(*
============================================================
PROGRAM: MAIN
============================================================

PURPOSE
  Top-level program that orchestrates all function blocks
  and manages the system data bus between GVLs.

EXECUTION ORDER (every PLC cycle)
  1. Initialise MQTT config from defaults (first scan only)
  2. Copy HMI inputs to GVL_System bus
  3. FB_SensorIO      — Read and scale analog sensor inputs
  4. FB_ValveControl  — Per-valve TC2_MC2 state machines (x3)
  5. Build timestamp string for MQTT and logging
  6. FB_MqttManager   — MQTT connection, publish, subscribe
  7. FB_CsvLogger     — Periodic CSV row logging
  8. Mirror runtime data to GVL_HMI for display
  9. Compute system health flags

DATA FLOW
  GVL_IO  --> FB_SensorIO --> GVL_System.Sensors
  GVL_HMI.HMI_* --> GVL_System.Valve[n] setpoints
  FB_MqttManager.rMqttValveSetpoint --> FB_ValveControl MQTT_Setpoint
  FB_ValveControl outputs --> GVL_System.Valve[n] status
  GVL_System.* --> GVL_HMI.ACT_* (for display)
  GVL_System.Valve + Sensors --> FB_MqttManager (outgoing JSON)
  GVL_System.Valve + Sensors --> FB_CsvLogger (CSV row)

LIBRARIES
  TC2_MC2, TF6701 / Tc3_IotBase, Tc2_System
============================================================
*)

PROGRAM MAIN
VAR
    // ── Function block instances ────────────────────────────────
    fbSensorIO      : FB_SensorIO;    //////Not Implemented currently
    fbValve1        : FB_ValveControl;
    fbValve2        : FB_ValveControl;
    fbValve3        : FB_ValveControl;
    fbCsvLogger     : FB_CsvLogger;
    fbMqttManager   : FB_MqttManager;

    // ── NC Axis references ──────────────────────────────────────
    // Each must be linked to an NC axis in TwinCAT I/O mapping.
    Axis_Valve1     : AXIS_REF;
    Axis_Valve2     : AXIS_REF;
    Axis_Valve3     : AXIS_REF;

    // ── Timestamp for MQTT JSON ──────────────────────────────────
    fbSysTime       : FB_LocalSystemTime;
    sTimestamp      : STRING(64);
    sTempStr        : STRING(8);

    // ── Whole-array buffers passed to FB_MqttManager ─────────────
    // TwinCAT does not allow per-element array assignment inside
    // an FB call's parameter list. Populate these arrays each
    // cycle, then pass them in a single assignment.
    aValveSetpoint  : ARRAY[1..3] OF REAL;
    aValveActual    : ARRAY[1..3] OF REAL;
    aValveSource    : ARRAY[1..3] OF STRING(8);

    // ── First-scan flag for MQTT default config load ─────────────
    bMqttConfigInit : BOOL := FALSE;
END_VAR

// ============================================================
// STEP 0 — ONE-TIME INITIALISATION
// On first scan, copy MQTT defaults from GVL_Config into the
// HMI-bound config struct. The operator can then edit any field
// from the HMI MQTT panel and click Apply to reconnect.
// ============================================================
IF NOT bMqttConfigInit THEN
    GVL_HMI.HMI_MQTT_Config.sBrokerAddress         := GVL_Config.MQTT_DEFAULT_BROKER_IP;
    GVL_HMI.HMI_MQTT_Config.nPort                  := GVL_Config.MQTT_DEFAULT_PORT;
    GVL_HMI.HMI_MQTT_Config.sClientId              := GVL_Config.MQTT_DEFAULT_CLIENT_ID;
    GVL_HMI.HMI_MQTT_Config.sUsername              := GVL_Config.MQTT_DEFAULT_USERNAME;
    GVL_HMI.HMI_MQTT_Config.sPassword              := GVL_Config.MQTT_DEFAULT_PASSWORD;
    GVL_HMI.HMI_MQTT_Config.sTopicPrefix           := GVL_Config.MQTT_DEFAULT_TOPIC_PREFIX;
    GVL_HMI.HMI_MQTT_Config.sMainTopic             := GVL_Config.MQTT_DEFAULT_MAIN_TOPIC;
    GVL_HMI.HMI_MQTT_Config.SubscribeTopic         := GVL_Config.MQTT_DEFAULT_SUB_TOPIC;
    GVL_HMI.HMI_MQTT_Config.tStatusPublishInterval := UDINT_TO_TIME(UINT_TO_UDINT(GVL_Config.MQTT_DEFAULT_PUBLISH_INTERVAL) * 1000);
    GVL_HMI.HMI_MQTT_Config.bUseStatusPublish      := TRUE;
   // bMqttConfigInit := TRUE;
END_IF


// ============================================================
// STEP 1 — COPY HMI SETPOINTS / RESETS INTO SYSTEM BUS
// ============================================================
GVL_System.Valve[1].HMI_Setpoint := GVL_HMI.HMI_Valve1_Setpoint;
GVL_System.Valve[1].Reset_Cmd    := GVL_HMI.HMI_Valve1_Reset;

GVL_System.Valve[2].HMI_Setpoint := GVL_HMI.HMI_Valve2_Setpoint;
GVL_System.Valve[2].Reset_Cmd    := GVL_HMI.HMI_Valve2_Reset;

GVL_System.Valve[3].HMI_Setpoint := GVL_HMI.HMI_Valve3_Setpoint;
GVL_System.Valve[3].Reset_Cmd    := GVL_HMI.HMI_Valve3_Reset;

// Reset-All button: propagate to all valves and self-clear
IF GVL_HMI.HMI_ResetAll THEN
    GVL_System.Valve[1].Reset_Cmd := TRUE;
    GVL_System.Valve[2].Reset_Cmd := TRUE;
    GVL_System.Valve[3].Reset_Cmd := TRUE;
    GVL_HMI.HMI_ResetAll := FALSE;
END_IF
// MQTT setpoints from FB_MqttManager (parsed from incoming JSON)
GVL_System.Valve[1].MQTT_Setpoint := fbMqttManager.rMqttValveSetpoint[1];
GVL_System.Valve[2].MQTT_Setpoint := fbMqttManager.rMqttValveSetpoint[2];
GVL_System.Valve[3].MQTT_Setpoint := fbMqttManager.rMqttValveSetpoint[3];
// Per-valve MQTT enable: master AND HMI checkbox AND command-level enable
GVL_System.Valve[1].MQTT_Enabled :=
    GVL_HMI.HMI_MQTT_bEnable AND
    GVL_HMI.HMI_Valve1_MQTT_Enable AND
    fbMqttManager.bMqttValveEnable[1];
GVL_System.Valve[2].MQTT_Enabled :=
    GVL_HMI.HMI_MQTT_bEnable AND
    GVL_HMI.HMI_Valve2_MQTT_Enable AND
    fbMqttManager.bMqttValveEnable[2];
GVL_System.Valve[3].MQTT_Enabled :=
    GVL_HMI.HMI_MQTT_bEnable AND
    GVL_HMI.HMI_Valve3_MQTT_Enable AND
    fbMqttManager.bMqttValveEnable[3];

// Active setpoint — diagnostic copy reflecting whatever the FB chose
GVL_System.Valve[1].Active_Setpoint := GVL_HMI.HMI_Valve1_Setpoint;
GVL_System.Valve[2].Active_Setpoint := GVL_HMI.HMI_Valve2_Setpoint;
GVL_System.Valve[3].Active_Setpoint := GVL_HMI.HMI_Valve3_Setpoint;


// ============================================================
// STEP 2 — SENSOR I/O
// Reads raw ADC, scales to engineering units, applies LPF.
// Must run before any FB that consumes GVL_System.Sensors.
// ============================================================
fbSensorIO(
    bEnable   := TRUE,
    rLpfAlpha := 0.1,           // 10 % new sample per cycle (moderate filtering)
    stOut     => GVL_System.Sensors
);


// ============================================================
// STEP 3 — VALVE 1
// ============================================================
fbValve1(
    Axis             := Axis_Valve1,
    HMI_Setpoint     := GVL_System.Valve[1].HMI_Setpoint,
    MQTT_Setpoint    := GVL_System.Valve[1].MQTT_Setpoint,
    MQTT_Enabled    := GVL_System.Valve[1].MQTT_Enabled,
    Enable           := TRUE,
    eHomingSelection := MC_DefaultHoming, //MC_Direct,
    Reset            := GVL_System.Valve[1].Reset_Cmd,
    Move_Stop        := GVL_HMI.HMI_Valve1_Stop,
    UPDATE           := GVL_HMI.HMI_UPDATE,
    ZeroPosition     := GVL_IO.bBottom_position_1,
	TopPosition		 := GVL_IO.bTop_position_1,  
    bHoming          := GVL_HMI.HMI_Valve1_Homing,
    MoveVelocity     := GVL_Config.VALVE_MOVE_VELOCITY,
    MoveAccel        := GVL_Config.VALVE_MOVE_ACCELERATION,
    MoveDecel        := GVL_Config.VALVE_MOVE_DECELERATION,
    MoveJerk         := GVL_Config.VALVE_MOVE_JERK,
    HomeVelocity     := GVL_Config.VALVE_HOMING_VELOCITY,
    FullStroke_mm    := GVL_Config.VALVE_FULL_STROKE_MM,
    PosTolerance     := GVL_Config.VALVE_POSITION_TOLERANCE,

    Actual_Position  => GVL_System.Valve[1].Actual_Position,
    State            => GVL_System.Valve[1].State,
    Source           => GVL_System.Valve[1].Source,
    IsHomed          => GVL_System.Valve[1].IsHomed,
    InPosition       => GVL_System.Valve[1].InPosition,
    IsFault          => GVL_System.Valve[1].IsFault,
    FaultCode        => GVL_System.Valve[1].FaultCode,
    rTarget_mm       => GVL_HMI.Raw_Valve1_Setpoint,
    rActual_mm       => GVL_HMI.Raw_Valve1_Position
);


// ============================================================
// STEP 4 — VALVE 2
// ============================================================
fbValve2(
    Axis             := Axis_Valve2,
    HMI_Setpoint     := GVL_System.Valve[2].HMI_Setpoint,
    MQTT_Setpoint    := GVL_System.Valve[2].MQTT_Setpoint,
    MQTT_Enabled    := GVL_System.Valve[2].MQTT_Enabled,
    Enable           := TRUE,
    eHomingSelection := MC_Direct,
    Reset            := GVL_System.Valve[2].Reset_Cmd,
    Move_Stop        := GVL_HMI.HMI_Valve2_Stop,
    UPDATE           := GVL_HMI.HMI_UPDATE,
    ZeroPosition     := GVL_IO.bBottom_position_1,   // Wire a separate limit switch per valve in HW
    bHoming          := GVL_HMI.HMI_Valve2_Homing,
    MoveVelocity     := GVL_Config.VALVE_MOVE_VELOCITY,
    MoveAccel        := GVL_Config.VALVE_MOVE_ACCELERATION,
    MoveDecel        := GVL_Config.VALVE_MOVE_DECELERATION,
    MoveJerk         := GVL_Config.VALVE_MOVE_JERK,
    HomeVelocity     := GVL_Config.VALVE_HOMING_VELOCITY,
    FullStroke_mm    := GVL_Config.VALVE_FULL_STROKE_MM,
    PosTolerance     := GVL_Config.VALVE_POSITION_TOLERANCE,

    Actual_Position  => GVL_System.Valve[2].Actual_Position,
    State            => GVL_System.Valve[2].State,
    Source           => GVL_System.Valve[2].Source,
    IsHomed          => GVL_System.Valve[2].IsHomed,
    InPosition       => GVL_System.Valve[2].InPosition,
    IsFault          => GVL_System.Valve[2].IsFault,
    FaultCode        => GVL_System.Valve[2].FaultCode,
    rTarget_mm       => GVL_HMI.Raw_Valve2_Setpoint,
    rActual_mm       => GVL_HMI.Raw_Valve2_Position
);


// ============================================================
// STEP 5 — VALVE 3
// ============================================================
fbValve3(
    Axis             := Axis_Valve3,
    HMI_Setpoint     := GVL_System.Valve[3].HMI_Setpoint,
    MQTT_Setpoint    := GVL_System.Valve[3].MQTT_Setpoint,
    MQTT_Enabled    := GVL_System.Valve[3].MQTT_Enabled,
    Enable           := TRUE,
    eHomingSelection := MC_Direct,
    Reset            := GVL_System.Valve[3].Reset_Cmd,
    Move_Stop        := GVL_HMI.HMI_Valve3_Stop,
    UPDATE           := GVL_HMI.HMI_UPDATE,
    ZeroPosition     := GVL_IO.bBottom_position_1,   // Wire a separate limit switch per valve in HW
    bHoming          := GVL_HMI.HMI_Valve3_Homing,
    MoveVelocity     := GVL_Config.VALVE_MOVE_VELOCITY,
    MoveAccel        := GVL_Config.VALVE_MOVE_ACCELERATION,
    MoveDecel        := GVL_Config.VALVE_MOVE_DECELERATION,
    MoveJerk         := GVL_Config.VALVE_MOVE_JERK,
    HomeVelocity     := GVL_Config.VALVE_HOMING_VELOCITY,
    FullStroke_mm    := GVL_Config.VALVE_FULL_STROKE_MM,
    PosTolerance     := GVL_Config.VALVE_POSITION_TOLERANCE,

    Actual_Position  => GVL_System.Valve[3].Actual_Position,
    State            => GVL_System.Valve[3].State,
    Source           => GVL_System.Valve[3].Source,
    IsHomed          => GVL_System.Valve[3].IsHomed,
    InPosition       => GVL_System.Valve[3].InPosition,
    IsFault          => GVL_System.Valve[3].IsFault,
    FaultCode        => GVL_System.Valve[3].FaultCode,
    rTarget_mm       => GVL_HMI.Raw_Valve3_Setpoint,
    rActual_mm       => GVL_HMI.Raw_Valve3_Position
);


// ============================================================
// STEP 6 — AUTO-CLEAR RESET COMMANDS
// Reset is edge-triggered inside FB_ValveControl, so clear here
// to prevent re-trigger on subsequent cycles.
// ============================================================
GVL_System.Valve[1].Reset_Cmd := FALSE;
GVL_HMI.HMI_Valve1_Reset      := FALSE;
GVL_System.Valve[2].Reset_Cmd := FALSE;
GVL_HMI.HMI_Valve2_Reset      := FALSE;
GVL_System.Valve[3].Reset_Cmd := FALSE;
GVL_HMI.HMI_Valve3_Reset      := FALSE;


// ============================================================
// STEP 7 — BUILD TIMESTAMP STRING (YYYY-MM-DD HH:MM:SS)
// Used for MQTT JSON and CSV row timestamps.
// ============================================================
(*fbSysTime(bEnable := TRUE, dwCycle := 1);

sTimestamp := UINT_TO_STRING(fbSysTime.systemTime.wYear);
sTimestamp := CONCAT(sTimestamp, '-');
sTempStr   := UINT_TO_STRING(fbSysTime.systemTime.wMonth);
IF fbSysTime.systemTime.wMonth < 10 THEN sTempStr := CONCAT('0', sTempStr); END_IF
sTimestamp := CONCAT(sTimestamp, sTempStr);
sTimestamp := CONCAT(sTimestamp, '-');
sTempStr   := UINT_TO_STRING(fbSysTime.systemTime.wDay);
IF fbSysTime.systemTime.wDay < 10 THEN sTempStr := CONCAT('0', sTempStr); END_IF
sTimestamp := CONCAT(sTimestamp, sTempStr);
sTimestamp := CONCAT(sTimestamp, ' ');
sTempStr   := UINT_TO_STRING(fbSysTime.systemTime.wHour);
IF fbSysTime.systemTime.wHour < 10 THEN sTempStr := CONCAT('0', sTempStr); END_IF
sTimestamp := CONCAT(sTimestamp, sTempStr);
sTimestamp := CONCAT(sTimestamp, ':');
sTempStr   := UINT_TO_STRING(fbSysTime.systemTime.wMinute);
IF fbSysTime.systemTime.wMinute < 10 THEN sTempStr := CONCAT('0', sTempStr); END_IF
sTimestamp := CONCAT(sTimestamp, sTempStr);
sTimestamp := CONCAT(sTimestamp, ':');
sTempStr   := UINT_TO_STRING(fbSysTime.systemTime.wSecond);
IF fbSysTime.systemTime.wSecond < 10 THEN sTempStr := CONCAT('0', sTempStr); END_IF
sTimestamp := CONCAT(sTimestamp, sTempStr);
*)

// ============================================================
// STEP 8 — MQTT MANAGER
// Populate whole-array buffers (per-element assignment is not
// allowed inside an FB call), then run the manager.
// ============================================================

// Build the array buffers required by FB_MqttManager
aValveSetpoint[1] := GVL_System.Valve[1].Active_Setpoint;
aValveSetpoint[2] := GVL_System.Valve[2].Active_Setpoint;
aValveSetpoint[3] := GVL_System.Valve[3].Active_Setpoint;

aValveActual[1] := GVL_System.Valve[1].Actual_Position;
aValveActual[2] := GVL_System.Valve[2].Actual_Position;
aValveActual[3] := GVL_System.Valve[3].Actual_Position;

aValveSource[1] := GVL_HMI.ACT_Valve1_SourceText;
aValveSource[2] := GVL_HMI.ACT_Valve2_SourceText;
aValveSource[3] := GVL_HMI.ACT_Valve3_SourceText;

fbMqttManager(
    bEnable              := GVL_HMI.HMI_MQTT_bEnable,
    stConfig             := GVL_HMI.HMI_MQTT_Config,
    bApplyConfig         := GVL_HMI.HMI_MQTT_ApplyConfig,
    bPublish             := GVL_HMI.HMI_MQTT_mPublish,
    bEnableStatusPublish := GVL_HMI.HMI_MQTT_Config.bUseStatusPublish,
    tStatusPublishTime   := GVL_HMI.HMI_MQTT_Config.tStatusPublishInterval,
    sStatusTopic         := GVL_HMI.HMI_MQTT_Config.sMainTopic,

    rValveSetpoint       := aValveSetpoint,
    rValveActual         := aValveActual,
    sValveSource         := aValveSource,

    rTemperature_C       := GVL_System.Sensors.rTemperature_C[1],
    rWaterLevel_pct      := GVL_System.Sensors.rWaterLevel_pct,
    rWaterLevel_mm       := GVL_System.Sensors.rWaterLevel_mm,
    sTimestamp           := sTimestamp,

    bConnected           => GVL_System.MQTT_Connected,
    bError               => GVL_System.MQTT_Error,
    nErrorCode           => GVL_System.MQTT_LastErrorCode,
    sErrorMsg            => GVL_System.MQTT_LastErrorMsg,
    sLastRxTopic         => GVL_System.MQTT_LastRxTopic,
    sLastRxPayload       => GVL_System.MQTT_LastRxPayload,
    sJsonStatusPayload   => GVL_System.MQTT_LastJsonStatus,
    bNewRemoteCommand    => GVL_System.MQTT_NewCommand,
	
	LastmsgPub			=> GVL_HMI.ACT_MQTT_LastMsgPubTime,
	LastmsgRcv 			=> GVL_HMI.ACT_MQTT_LastMsgRcvTime,
	currentState		=> GVL_HMI.ACT_MQTT_State
);

// Auto-clear Apply button after one cycle (rising edge consumed inside FB)
GVL_HMI.HMI_MQTT_ApplyConfig := FALSE;


// ============================================================
// STEP 9 — CSV LOGGER
// ============================================================
fbCsvLogger(
    bEnable          := GVL_HMI.HMI_CSV_Enable,
    bForceWrite      := GVL_HMI.WriteTrigger,
    tLogInterval     := GVL_Config.CSV_LOG_INTERVAL_S,
    sBasePath        := GVL_Config.CSV_FILE_PATH,
    sPrefix          := GVL_Config.CSV_FILENAME_PREFIX,
    stValve          := GVL_System.Valve,
    stSensors        := GVL_System.Sensors,

    dtLastWrite      => GVL_System.CSV_LastWriteTime,
    bError           => GVL_System.CSV_FileError,
    sCurrentFilename => GVL_System.CSV_CurrentFile,
    eState           => GVL_System.CSV_LoggerState
);

// Auto-clear write trigger after one cycle
GVL_HMI.WriteTrigger := FALSE;


// ============================================================
// STEP 10 — MIRROR FEEDBACK TO HMI DISPLAY VARIABLES
// All ACT_* variables are read-only from the HMI side.
// ============================================================

// Valve 1 feedback
GVL_HMI.ACT_Valve1_Position  := GVL_System.Valve[1].Actual_Position;
GVL_HMI.ACT_Valve1_State     := GVL_System.Valve[1].State;
GVL_HMI.ACT_Valve1_Source    := GVL_System.Valve[1].Source;
GVL_HMI.ACT_Valve1_Fault     := GVL_System.Valve[1].IsFault;
GVL_HMI.ACT_Valve1_FaultCode := GVL_System.Valve[1].FaultCode;

// Valve 2 feedback
GVL_HMI.ACT_Valve2_Position  := GVL_System.Valve[2].Actual_Position;
GVL_HMI.ACT_Valve2_State     := GVL_System.Valve[2].State;
GVL_HMI.ACT_Valve2_Source    := GVL_System.Valve[2].Source;
GVL_HMI.ACT_Valve2_Fault     := GVL_System.Valve[2].IsFault;
GVL_HMI.ACT_Valve2_FaultCode := GVL_System.Valve[2].FaultCode;

// Valve 3 feedback
GVL_HMI.ACT_Valve3_Position  := GVL_System.Valve[3].Actual_Position;
GVL_HMI.ACT_Valve3_State     := GVL_System.Valve[3].State;
GVL_HMI.ACT_Valve3_Source    := GVL_System.Valve[3].Source;
GVL_HMI.ACT_Valve3_Fault     := GVL_System.Valve[3].IsFault;
GVL_HMI.ACT_Valve3_FaultCode := GVL_System.Valve[3].FaultCode;

// Source text strings (HMI indicators + MQTT JSON sValveSource[])
CASE GVL_System.Valve[1].Source OF
    E_ValveSource.MQTT: GVL_HMI.ACT_Valve1_SourceText := 'MQTT';
    E_ValveSource.HMI:  GVL_HMI.ACT_Valve1_SourceText := 'HMI';
    ELSE                GVL_HMI.ACT_Valve1_SourceText := 'NONE';
END_CASE

CASE GVL_System.Valve[2].Source OF
    E_ValveSource.MQTT: GVL_HMI.ACT_Valve2_SourceText := 'MQTT';
    E_ValveSource.HMI:  GVL_HMI.ACT_Valve2_SourceText := 'HMI';
    ELSE                GVL_HMI.ACT_Valve2_SourceText := 'NONE';
END_CASE

CASE GVL_System.Valve[3].Source OF
    E_ValveSource.MQTT: GVL_HMI.ACT_Valve3_SourceText := 'MQTT';
    E_ValveSource.HMI:  GVL_HMI.ACT_Valve3_SourceText := 'HMI';
    ELSE                GVL_HMI.ACT_Valve3_SourceText := 'NONE';
END_CASE

// Sensor displays
GVL_HMI.ACT_WaterLevel_pct  := GVL_System.Sensors.rWaterLevel_pct;
GVL_HMI.ACT_WaterLevel_mm   := GVL_System.Sensors.rWaterLevel_mm;
GVL_HMI.ACT_Temperature1_C  := GVL_System.Sensors.rTemperature_C[1];
GVL_HMI.ACT_Temperature2_C  := GVL_System.Sensors.rTemperature_C[2];
GVL_HMI.ACT_SensorFault     := GVL_System.Sensors.bAnySensorFault;

// MQTT status
GVL_HMI.ACT_MQTT_Connected   := GVL_System.MQTT_Connected;
GVL_HMI.ACT_MQTT_Error       := GVL_System.MQTT_Error;
GVL_HMI.ACT_MQTT_ErrorMsg    := GVL_System.MQTT_LastErrorMsg;
GVL_HMI.ACT_MQTT_JsonPreview := GVL_System.MQTT_LastJsonStatus;
GVL_HMI.ACT_MQTT_LastRxTopic := GVL_System.MQTT_LastRxTopic;
GVL_HMI.ACT_MQTT_NewCommand  := GVL_System.MQTT_NewCommand;

// CSV status
GVL_HMI.ACT_CSV_CurrentFile   := GVL_System.CSV_CurrentFile;
GVL_HMI.ACT_CSV_LastWriteTime := GVL_System.CSV_LastWriteTime;
GVL_HMI.ACT_CSV_Error         := GVL_System.CSV_FileError;


// ============================================================
// STEP 11 — SYSTEM HEALTH FLAGS
// ============================================================
GVL_System.AnyFaultActive :=
    GVL_System.Valve[1].IsFault OR
    GVL_System.Valve[2].IsFault OR
    GVL_System.Valve[3].IsFault;

GVL_System.AnySensorFault := GVL_System.Sensors.bAnySensorFault;

GVL_System.SystemReady :=
    GVL_System.Valve[1].IsHomed AND
    GVL_System.Valve[2].IsHomed AND
    GVL_System.Valve[3].IsHomed AND
    NOT GVL_System.AnyFaultActive;

GVL_HMI.ACT_SystemReady := GVL_System.SystemReady;

END_PROGRAM

(* stored: Version 1.1.0.1, ProductVersion 3.1.4026.18
   POU MAIN: Id {a0f99a09-eccb-42d8-b9bd-167b13d45a91}, SpecialFunc None *)
